// TIA Portal V19 export
FUNCTION_BLOCK "TYPIC_C403_IF_LVE"   // FB132, FBD
TITLE = TYPIC_C403_IF_LVE: Detectiepunt
{ S7_Optimized_Access := 'TRUE' }
AUTHOR : OCOTECH
FAMILY : Typical
NAME : C403.702
// Logisch Object Besturing: C403.701
// 
// Het doel van de IF LVE (Detectiepunt SnelheidsOnderschrijding) is om de gegevens te verwerken die ontvangen worden van een detectiepunt uit de interne sturing en via inputs.
// stored: MemoryReserve 10, SetENOAutomatically false
   VAR_INPUT
      EXT_HW { ExternalAccessible := 'False'; ExternalVisible := 'False'; ExternalWritable := 'False'} : Bool;   // Sturings hardware (PLC) bewaking (1 = OK)
      IN_AUT_C403 { ExternalAccessible := 'False'; ExternalVisible := 'False'; ExternalWritable := 'False'} : Bool;   // Beveiligingen: serie geschakelde terugmelding (1= OK)
      IN_AUT { ExternalAccessible := 'False'; ExternalVisible := 'False'; ExternalWritable := 'False'} : Bool;   // Beveiliging kastklimatisatie (1 = OK)
      IN_SPD_OK { ExternalAccessible := 'False'; ExternalVisible := 'False'; ExternalWritable := 'False'} : Bool;   // Status overspanningsbeveiliging (1 = OK)
      IN_DEC { ExternalAccessible := 'False'; ExternalVisible := 'False'; ExternalWritable := 'False'} : Bool;   // Deurcontact (1 = Gesloten)
      IN_STS { ExternalAccessible := 'False'; ExternalVisible := 'False'; ExternalWritable := 'False'} : Word;   // Statusbits van een lusdetectie
   END_VAR
   VAR_OUTPUT
      VAR_IF_LVE { ExternalAccessible := 'False'; ExternalVisible := 'False'; ExternalWritable := 'False'} : "C403_VAR_IF_LVE_TYPIC";   // Struct met alle variabelen naar de subfunctie
   END_VAR
   VAR
      STO { ExternalWritable := 'False'} : Struct   // Storingen
         A001 : Bool;   // Beveiliging aangesproken
         A002 : Bool;   // Storing detectiepunt
         A003 : Bool;   // Beveiliging klimaatregeling wegkantkast aangesproken
         A004 : Bool;   // Overspanningsbeveiliging aangesproken
      END_STRUCT;
      VAR { ExternalWritable := 'False'} : Struct   // Variabelen
         EXT_HW { ExternalAccessible := 'False'; ExternalVisible := 'False'} : Bool;   // Sturings hardware (PLC) in storing
         STS_KST_OPEN { ExternalAccessible := 'False'; ExternalVisible := 'False'} : Bool;   // TRUE = deur wegkantkast geopend
         STS_NEG { ExternalAccessible := 'False'; ExternalVisible := 'False'} : Bool;   // Spookrijder gedetecteerd
         STS_SOS { ExternalAccessible := 'False'; ExternalVisible := 'False'} : Bool;   // Snelheidsonderschrijding
         STS_STOP { ExternalAccessible := 'False'; ExternalVisible := 'False'} : Bool;   // Stilstand
      END_STRUCT;
   END_VAR
BEGIN

REGION Network 1: START
END_REGION

REGION Network 2: +++ Verkeersstatus +++
   // De door het detectiepunt geregistreerde verkeersstatus wordt doorgegeven aan 3B.
END_REGION

REGION Network 3: +++ Bewaking deur wegkantkast +++
   // De bewaking van de deur van de wegkantkast is enkel van toepassing voor detectiepunten die zich buiten de verkeerskoker bevinden en die aangesloten zijn via een wegkantkast behorende tot deelsysteem C403 (SOS).
END_REGION

REGION Network 4: +++ Storingen +++
   // Verzamelen storingsmeldingen.
END_REGION

REGION Network 5: Storing A001: Beveiliging aangesproken
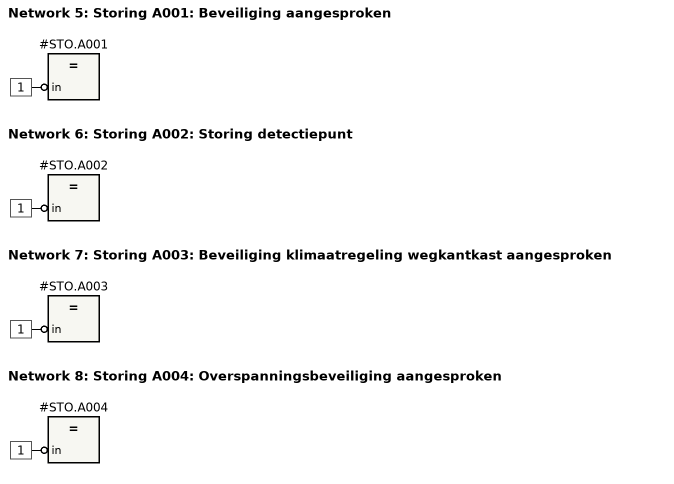
   #STO.A001 := NOT 1;
END_REGION

REGION Network 6: Storing A002: Storing detectiepunt
   #STO.A002 := NOT 1;
END_REGION

REGION Network 7: Storing A003: Beveiliging klimaatregeling wegkantkast aangesproken
   #STO.A003 := NOT 1;
END_REGION

REGION Network 8: Storing A004: Overspanningsbeveiliging aangesproken
   #STO.A004 := NOT 1;
END_REGION

REGION Network 9 (SCL): EINDE
   // Variabelen van intern scada rakvlak naar outputs copieren
   #VAR_IF_LVE.EXT_HW := #VAR.EXT_HW;
   #VAR_IF_LVE.STS_KST_OPEN := #VAR.STS_KST_OPEN;
   #VAR_IF_LVE.STS_NEG := #VAR.STS_NEG;
   #VAR_IF_LVE.STS_SOS := #VAR.STS_SOS;
   #VAR_IF_LVE.STS_STOP := #VAR.STS_STOP;
   #VAR_IF_LVE.STO := #STO;
END_REGION
END_FUNCTION_BLOCK
